// TIA Portal V20 export
TYPE "typeEm7MonitoringJobInterface"
// stored: Access Published, Namespace Unit1
   STRUCT
      busySTK1QrRead { ExternalWritable := 'False'} : Bool;
      doneSTK1QrRead { ExternalWritable := 'False'} : Bool;
      busySTK2QrRead { ExternalWritable := 'False'} : Bool;
      doneSTK2QrRead { ExternalWritable := 'False'} : Bool;
   END_STRUCT;
END_TYPE
